# EPICS autosave request: iocBoot/iocnv40/auto_settings.req
file motor_settings.req P=NV40:,M=ax1
file motor_settings.req P=NV40:,M=ax2
file motor_settings.req P=NV40:,M=ax3
